Yaskawa INFORM job: SKRZYNIA_5340_90_STOPNI_20BR_OLD.JBI

/JOB
//NAME SKRZYNIA_5340_90_STOPNI_20BR_OLD
///FOLDERNAME 02-SKRZYNIE_JOBS
//POS
///NPOS 552,552,0,39,0,0
///TOOL 0
///POSTYPE PULSE
///PULSE
C00000=0,-52280,40443,0,6876,0
C00001=82314,-24956,17040,59626,-27382,6248
C00002=93910,-8625,17040,59626,-43355,6248
C00003=98846,-1061,-42166,80308,-57081,-16120
C00004=100452,6057,-48127,85711,-56704,-21322
C00005=95573,33077,-33257,84645,-64023,-26851
C00006=94102,33899,-31937,85246,-63371,-26689
C00007=95573,33077,-33257,84645,-64023,-26851
C00008=94862,31071,-36438,85313,-63677,-27192
C00009=95573,33077,-33257,84645,-64023,-26851
C00010=95263,33142,-33256,84677,-63995,-26850
C00011=95263,33142,-33256,84677,-63995,-26850
C00012=94017,33843,-32133,85187,-63445,-26710
C00013=95557,35310,-29762,82906,-65354,-26497
C00014=95275,35582,-29321,82044,-66131,-26480
C00015=95263,33142,-33256,84677,-63995,-26850
C00016=95260,33144,-33256,84678,-63995,-26850
C00017=95260,33144,-33256,84678,-63995,-26850
C00018=94022,33838,-32141,85183,-63448,-26711
C00019=95260,33144,-33256,84678,-63995,-26850
C00020=94618,31343,-36117,85281,-63684,-27157
C00021=95260,33144,-33256,84678,-63995,-26850
C00022=95258,25631,32269,66559,-75499,-2416
C00023=95258,25631,32269,66559,-75499,-2416
C00024=94181,26497,33533,66410,-74896,-2191
C00025=95658,30184,39035,66708,-78559,-2356
C00026=95217,30377,39331,66881,-79841,-2558
C00027=95258,25631,32269,66559,-75499,-2416
C00028=98811,21047,-15512,99242,-81394,-20987
C00029=98811,21047,-15512,99242,-81394,-20987
C00030=97775,21639,-14693,99563,-80753,-20993
C00031=98811,21047,-15512,99242,-81394,-20987
C00032=98206,18840,-18520,99489,-81124,-21211
C00033=98811,21047,-15512,99242,-81394,-20987
C00034=98765,34858,63506,90961,-74847,-417
C00035=98765,34858,63506,90961,-74847,-417
C00036=97741,35895,65220,90657,-74158,-246
C00037=98765,34858,63506,90961,-74847,-417
C00038=98337,32226,59232,91111,-74633,-884
C00039=98765,34858,63506,90961,-74847,-417
C00040=98728,21792,17445,103800,-78809,-12049
C00041=97232,27021,37502,101932,-75086,-7690
C00042=96358,27701,38514,101868,-74464,-7680
C00043=97232,27021,37502,101932,-75086,-7690
C00044=96733,24820,34282,102049,-74905,-7989
C00045=97232,27021,37502,101932,-75086,-7690
C00046=94428,854,16076,89248,-50738,-4740
C00047=88080,-20128,-3199,80943,-31244,-2335
C00048=48287,-44591,-17414,16172,-14532,25809
C00049=48287,-44591,-17414,16172,-14532,25809
C00050=85348,-13130,13838,41209,-47455,8220
C00051=97395,20012,29210,69700,-74457,-9077
C00052=97055,28839,36684,71776,-79389,-10554
C00053=97055,28839,36684,71776,-79389,-10554
C00054=96058,29646,37897,71666,-78799,-10362
C00055=97055,28839,36684,71776,-79389,-10554
C00056=96570,26659,33451,71832,-78911,-10777
C00057=97055,28839,36684,71776,-79389,-10554
C00058=99123,23256,18377,81563,-78104,3156
C00059=99123,23256,18377,81563,-78104,3156
C00060=98123,23909,19300,81582,-77442,3256
C00061=99123,23256,18377,81563,-78104,3156
C00062=98765,21723,16234,81638,-77830,3017
C00063=99123,23256,18377,81563,-78104,3156
C00064=99222,23346,17795,82202,-78388,4176
C00065=99222,23346,17795,82202,-78388,4176
C00066=98149,24045,18779,82229,-77677,4281
C00067=99222,23346,17795,82202,-78388,4176
C00068=98861,21801,15633,82278,-78114,4033
C00069=99222,23346,17795,82202,-78388,4176
C00070=100468,18781,12295,88713,-76630,3899
C00071=100488,13084,3722,91602,-74275,2573
C00072=99329,-2479,-35949,113241,-72472,-2557
C00073=60067,-64368,-72505,144806,-26050,-19168
C00074=60067,-50244,-32501,110603,-14199,-2207
C00075=63330,-26972,24478,18707,-56801,31483
C00076=95462,-32664,-40336,69376,-39980,4046
C00077=97787,-9790,-26685,81509,-54738,-4408
C00078=99864,21793,7359,80466,-76601,-6182
C00079=99862,21793,7358,80466,-76600,-6182
C00080=98290,21024,6297,80683,-75539,-6194
C00081=97471,21541,7008,80756,-75007,-6115
C00082=98290,21024,6297,80683,-75539,-6194
C00083=97834,19245,3873,80814,-75197,-6333
C00084=98290,21024,6297,80683,-75539,-6194
C00085=98946,26804,31705,85784,-78857,-1423
C00086=98946,26804,31705,85784,-78857,-1423
C00087=98292,27270,32391,85749,-78414,-1361
C00088=98946,26804,31705,85784,-78857,-1423
C00089=98631,25349,29587,85839,-78632,-1590
C00090=98946,26804,31705,85784,-78857,-1423
C00091=97031,6331,9149,87487,-63868,-1924
C00092=73503,-30722,-22703,70949,-18863,5788
C00093=42754,-66126,12236,-1301,3231,7194
C00094=0,-52280,40443,0,6876,0
C00095=0,-52280,40443,0,6876,0
C00096=48041,-29633,723,44271,-15597,-57965
C00097=50268,-18118,11295,51661,-15759,-61288
C00098=49280,-17155,12057,50642,-15139,-60911
C00099=50435,-16984,12194,52574,-15707,-61719
C00100=49536,-18455,11034,50297,-15435,-60714
C00101=49756,-19891,11927,46282,-16637,-58724
C00102=49756,-15074,24021,36925,-20097,-54095
C00103=49264,-12389,27117,35970,-20004,-53698
C00104=48191,-11316,28046,34492,-19486,-53134
C00105=50556,-10584,28692,38442,-20269,-54728
C00106=49756,-15074,24021,36925,-20097,-54095
C00107=50509,-14376,22441,40930,-19158,-55976
C00108=50873,-17966,11417,52677,-16048,-61710
C00109=49459,-16590,12517,51258,-15158,-61190
C00110=50592,-16429,12648,53120,-15720,-61960
C00111=50873,-17966,11417,52677,-16048,-61710
C00112=50703,-18403,11066,52155,-16024,-61477
C00113=50703,-18403,11066,52155,-16024,-61477
C00114=49026,-16768,12358,50435,-14971,-60844
C00115=50653,-16371,12680,53228,-15754,-62008
C00116=50703,-18403,11066,52155,-16024,-61477
C00117=50704,-18401,11069,52157,-16021,-61478
C00118=50704,-20525,5414,58956,-14779,-64789
C00119=49025,-18889,6668,57745,-13658,-64384
C00120=50799,-18420,7036,60610,-14610,-65581
C00121=50704,-20525,5414,58956,-14779,-64789
C00122=51005,-17995,11387,52847,-16122,-61778
C00123=51005,-17995,11387,52847,-16122,-61778
C00124=49564,-16598,12501,51417,-15218,-61257
C00125=50954,-16306,12737,53719,-15902,-62212
C00126=51005,-17995,11387,52847,-16122,-61778
C00127=51030,-17981,11395,52891,-16138,-61796
C00128=51030,-17981,11395,52891,-16138,-61796
C00129=49401,-16396,12662,51265,-15114,-61201
C00130=50908,-16047,12947,53789,-15850,-62250
C00131=51030,-17981,11395,52891,-16138,-61796
C00132=50945,-18019,11363,52741,-16103,-61737
C00133=50945,-16980,14081,49884,-16761,-60338
C00134=49117,-15186,15539,47848,-15653,-59576
C00135=50939,-14679,15960,50992,-16487,-60881
C00136=50945,-18019,11363,52741,-16103,-61737
C00137=50945,-18019,11363,52741,-16103,-61737
C00138=50945,-18556,9943,54337,-15776,-62517
C00139=48967,-16606,11493,52445,-14510,-61829
C00140=51083,-15952,12027,56053,-15559,-63336
C00141=50945,-18556,9943,54337,-15776,-62517
C00142=50945,-18019,11363,52741,-16103,-61737
C00143=51350,-15183,18375,46705,-17991,-58719
C00144=49319,-13187,20053,44263,-16830,-57796
C00145=51236,-12618,20544,47529,-17647,-59142
C00146=51350,-15183,18375,46705,-17991,-58719
C00147=50028,-23690,-6096,22921,-31075,-54538
C00148=50670,-23735,-6923,24003,-30760,-55076
C00149=48518,-21492,-5254,21861,-29696,-54082
C00150=50138,-21068,-4928,23831,-30039,-55022
C00151=50670,-23735,-6923,24003,-30760,-55076
C00152=49763,-24225,-29961,22080,-30065,-59113
C00153=49763,-24225,-29961,22080,-30065,-59113
C00154=47727,-21550,-27874,20313,-29013,-58119
C00155=49271,-21042,-27466,22016,-29310,-59069
C00156=49763,-24225,-29961,22080,-30065,-59113
C00157=50713,-12366,-58367,41124,-17813,-74400
C00158=50713,-12366,-58367,41124,-17813,-74400
C00159=48934,-9522,-55687,39981,-16902,-73526
C00160=50242,-8975,-55157,41389,-17374,-74448
C00161=50713,-12366,-58367,41124,-17813,-74400
C00162=49763,-25421,-36239,24565,-26935,-60445
C00163=43547,-31626,-19626,5157,-49140,-52118
C00164=40154,-51179,-915,24203,-8234,-36524
C00165=0,-52280,40443,0,6876,0
C00166=0,-52280,40443,0,6876,0
C00167=2117,-50103,-33543,4117,45077,-85249
C00168=-26439,-48928,-33543,4117,-52362,-85249
C00169=-1453,-29933,-32011,46693,-66666,-90474
C00170=24798,-19255,-10490,69050,-85424,-90395
C00171=18386,-22028,-12683,68302,-81515,-89477
///LIMIT ON
C00172=9843,-31743,-57176,61611,-65235,-99401
C00173=-39603,-23393,-71448,91573,-31907,-107123
C00174=-35705,5077,-63140,100511,-35979,-118164
C00175=-33789,12193,-59259,102607,-37482,-119984
C00176=-34998,13124,-58049,103267,-36945,-119997
C00177=-34401,14597,-56112,102586,-37131,-119778
C00178=-34998,13124,-58049,103267,-36945,-119997
C00179=-36388,13885,-57049,104079,-36338,-120048
C00180=-34998,13124,-58049,103267,-36945,-119997
C00181=-34008,-7969,-75285,118537,-50852,-116988
C00182=-26318,8527,-57077,128458,-81874,-108613
///LIMIT OFF
C00183=-23139,-1795,-12064,73373,-53703,-87448
C00184=-27830,-667,-10848,73187,-50621,-86997
C00185=-27373,916,-9115,73207,-50922,-87041
C00186=-27830,-667,-10848,73187,-50621,-86997
C00187=-28901,-207,-10348,73132,-49918,-86888
C00188=-27830,-667,-10848,73187,-50621,-86997
C00189=-37166,8347,13175,41366,-53536,-76331
C00190=-37403,7707,12401,41298,-53388,-76282
C00191=-36830,9273,14303,41455,-53750,-76396
C00192=-37403,7707,12401,41298,-53388,-76282
C00193=-38235,8246,13056,40951,-53040,-76025
C00194=-37403,7707,12401,41298,-53388,-76282
C00195=-30063,5992,18551,55847,-56234,-77619
C00196=-30754,7414,19761,55747,-55713,-77591
C00197=-30376,8670,21285,55817,-55984,-77619
C00198=-30754,7414,19761,55747,-55713,-77591
C00199=-31265,7672,20073,55566,-55435,-77478
C00200=-30085,6037,18588,55845,-56218,-77619
C00201=-25385,-1715,-9470,94765,-53990,-89712
C00202=-25885,-764,-8323,94779,-53645,-89697
C00203=-25564,418,-7032,94741,-53861,-89683
C00204=-25885,-764,-8323,94779,-53645,-89697
C00205=-26741,-428,-7957,94890,-53068,-89741
C00206=-25421,-1648,-9389,94767,-53966,-89710
C00207=-17789,-39335,-40320,90232,-41783,-86178
C00208=-25885,-761,-8324,94780,-53645,-89696
C00209=-25885,-761,-8324,94780,-53645,-89696
C00210=-25612,239,-7230,94748,-53828,-89684
C00211=-25885,-761,-8324,94780,-53645,-89696
C00212=-26712,-436,-7972,94885,-53087,-89742
C00213=-25885,-761,-8324,94780,-53645,-89696
C00214=-26038,-1317,-8919,94796,-53541,-89701
C00215=-18430,-29121,-33898,93348,-44706,-88207
C00216=-3209,-48313,-44409,84985,-37126,-83197
C00217=-3617,-53456,-46461,81793,-37023,-81323
C00218=-28991,-22310,-29554,94749,-46554,-89251
C00219=-30664,-6343,-14094,96248,-45630,-90223
C00220=-30664,-6343,-14094,96248,-45630,-90223
C00221=-30207,-5031,-12762,96238,-45949,-90236
C00222=-30664,-6343,-14094,96248,-45630,-90223
C00223=-31510,-5971,-13720,96406,-45066,-90297
C00224=-29506,-9179,-17232,96085,-46411,-90159
C00225=-30003,-8487,-16482,96169,-46079,-90194
C00226=-30881,-6301,-14053,96286,-45485,-90239
C00227=-30407,-4956,-12684,96275,-45813,-90252
C00228=-30881,-6301,-14053,96286,-45485,-90239
C00229=-31646,-5963,-13712,96429,-44974,-90305
C00230=-29893,-8752,-16772,96152,-46152,-90188
C00231=-30350,-7636,-15544,96220,-45845,-90215
C00232=-30881,-6301,-14053,96286,-45485,-90239
C00233=-30396,-4924,-12652,96275,-45822,-90251
C00234=-30881,-6301,-14053,96286,-45485,-90239
C00235=-31665,-5954,-13703,96434,-44961,-90308
C00236=-29959,-8593,-16598,96162,-46108,-90192
C00237=-26558,-19284,-27675,95285,-48332,-89713
C00238=-5136,-57382,-50746,80999,-31115,-81799
C00239=-5136,-57382,-50746,80999,-31115,-81799
C00240=-22762,-12288,-20025,94001,-55646,-89200
C00241=-24763,-3131,-11201,94769,-54426,-89746
C00242=-26203,-419,-7954,94818,-53430,-89712
C00243=-25939,548,-6896,94784,-53609,-89698
C00244=-26203,-419,-7954,94818,-53430,-89712
C00245=-26818,-174,-7689,94897,-53016,-89744
C00246=-24998,-2701,-10694,94780,-54264,-89743
C00247=-23275,-722,28392,94611,-50650,-77911
C00248=-21733,-16242,25206,75334,-39210,-63099
C00249=0,-52280,40443,0,6876,0
C00250=0,-52280,40443,0,6876,0
C00251=82314,-24956,17040,59626,-27382,6248
C00252=93910,-8625,17040,59626,-43355,6248
C00253=98846,-1061,-42166,80308,-57081,-16120
C00254=100452,6057,-48127,85711,-56704,-21322
C00255=95564,34698,-34234,85516,-63941,-27819
C00256=93687,36612,-31081,84292,-64733,-27467
C00257=93711,36598,-31105,84282,-64744,-27471
C00258=95564,34698,-34234,85516,-63941,-27819
C00259=96930,32282,-32252,82595,-65816,-26305
C00260=93663,32611,-31732,84127,-64318,-26195
C00261=93663,32611,-31732,84127,-64318,-26195
C00262=96930,32282,-32252,82595,-65816,-26305
C00263=96528,-7533,-34932,76119,-53878,-10439
C00264=88377,-34186,-45291,67238,-52212,-2442
C00265=73560,-62084,7826,28695,-34737,3666
C00266=0,-52280,40443,0,6876,0
C00267=0,-52280,40443,0,6876,0
C00268=2117,-50103,-33543,4117,45077,-85249
C00269=-26439,-48928,-33543,4117,-52362,-85249
C00270=-26439,-27355,-33543,41485,-52362,-85249
C00271=-39218,-24492,-41653,51934,-39374,-86964
C00272=-37997,-10433,-19136,70610,-34172,-88069
C00273=-38397,-8978,-17736,70703,-33874,-88109
C00274=-39218,-24492,-41653,51934,-39374,-86964
C00275=-26439,-27355,-33543,41485,-52362,-85249
C00276=1598,-24403,-16502,45671,-72599,-88798
C00277=-11365,-15171,10010,30164,-77975,-82960
C00278=-38112,4197,-14374,43778,-42973,-90436
C00279=-39116,7904,-10019,43942,-43580,-90646
C00280=-38495,8531,-9262,44482,-44499,-91194
C00281=-38112,4197,-14374,43778,-42973,-90436
C00282=-53220,-12364,-8957,19277,-47766,-73858
C00283=-11365,-15171,10010,30164,-77975,-82960
C00284=-16156,-38280,11293,23671,-42998,-42040
C00285=-11365,-47379,10010,30164,3063,-681
C00286=0,-52280,40443,0,6876,0
C00287=0,-36700,24612,-42871,-31823,-33862
C00288=44403,-30110,7154,24155,-23805,-45557
C00289=51347,-17798,16373,37641,-23556,-51399
C00290=51570,-17239,16856,38066,-23574,-51584
C00291=66077,-16287,3920,86568,-32028,-80947
C00292=60657,-14974,12588,70166,-26612,-71053
C00293=40431,-28773,9158,17648,-23273,-42875
C00294=0,-36700,24612,-42871,-31823,-33862
C00295=0,-52280,40443,0,6876,0
C00296=0,-52280,40443,0,6876,0
C00297=73560,-62084,7826,28695,-34737,3666
C00298=88377,-34186,-45291,67238,-52212,-2442
C00299=96528,-7533,-34932,76119,-53878,-10439
C00300=100432,21324,12575,83706,-77956,-7498
C00301=100432,21324,12575,83706,-77956,-7498
C00302=97224,21170,12361,83970,-75786,-7447
C00303=97224,21170,12361,83970,-75786,-7447
C00304=100432,21324,12575,83706,-77956,-7498
C00305=100432,21324,12575,83706,-77956,-7498
C00306=97481,25108,17890,83512,-78432,-7131
C00307=97624,25049,17805,83504,-78528,-7141
C00308=100432,21324,12575,83706,-77956,-7498
C00309=97137,1790,-11103,86179,-63102,-7963
C00310=99183,2264,5333,86781,-62651,-3264
C00311=99868,-33,22146,72719,-59601,5126
C00312=99028,-10516,17309,71061,-60695,4227
C00313=58820,-39124,10926,53325,-41870,3759
C00314=0,-52280,40443,0,6876,0
C00315=37281,-50778,-9546,79570,-75313,-71156
C00316=21038,-23698,-30323,82948,-81132,-85647
C00317=-27256,-5882,-14331,85818,-48304,-85968
C00318=-24751,2890,-4920,85349,-55822,-86178
C00319=-24793,2953,-4845,85351,-55796,-86173
C00320=-27256,-5882,-14331,85818,-48304,-85968
C00321=-21143,-15675,-23596,84785,-52496,-85466
C00322=35274,-15248,-23220,82440,-90817,-86704
C00323=35274,-15248,-23220,82440,-90817,-86704
C00324=-45551,161,-18089,35087,-36064,-73293
C00325=-42435,6767,-10562,40540,-41185,-77662
C00326=-42821,6494,-10882,40094,-40673,-77276
C00327=-45551,161,-18089,35087,-36064,-73293
C00328=-32891,-7184,-22739,69075,-41395,-83248
C00329=-29265,-39765,-39402,58096,-43152,-73226
C00330=-37287,-55159,35520,2191,5667,-2084
C00331=0,-52280,40443,0,6876,0
C00332=0,-36700,24612,-42871,-31823,-33862
C00333=44403,-30110,7154,24155,-23805,-45557
C00334=44403,-30110,7154,24155,-23805,-45557
C00335=42101,-12213,25656,103795,-5192,-78630
C00336=46259,-8171,27719,110365,-8144,-81138
C00337=52601,-3768,32601,101908,-15442,-75329
C00338=55043,-3560,27637,120535,-21833,-87376
C00339=55127,-3656,27536,120476,-21875,-87335
C00340=50677,-23266,8367,38735,-22212,-52049
C00341=47073,-34549,9488,27883,-30316,-51458
C00342=0,-52280,40443,0,6876,0
C00343=0,-52280,40443,0,6876,0
C00344=73560,-62084,7826,28695,-34737,3666
C00345=96983,-27116,-23481,78724,-62297,-1998
C00346=100467,-7393,-15195,81625,-60158,-6002
C00347=99336,18440,8642,84276,-74234,-7647
C00348=99336,18440,8642,84276,-74234,-7647
C00349=97735,24994,14595,85350,-78994,-5109
C00350=97744,25074,13580,86004,-79195,-4385
C00351=99336,18440,8642,84276,-74234,-7647
C00352=99336,18440,8642,84276,-74234,-7647
C00353=97891,23737,8261,88167,-79183,-2386
C00354=97851,23541,8142,88101,-79081,-2507
C00355=99336,18440,8642,84276,-74234,-7647
C00356=89817,-17341,-38408,97132,-45323,-12250
C00357=100347,-21961,-42251,93939,-52125,-11121
C00358=60204,-59872,-73451,117647,-17639,-18840
C00359=37721,-67612,11381,1325,-438,7850
C00360=-37287,-55159,35520,2191,5667,-2084
C00361=-40042,-68802,-18337,47708,-19461,-45384
C00362=-28646,-23138,-32952,89786,-42552,-85395
C00363=-38882,-16596,-17625,44304,-41043,-72768
C00364=-42680,-6319,-12818,46127,-36112,-73823
C00365=-37459,704,-5408,52536,-43357,-78192
C00366=-32778,4349,-7465,59128,-48375,-83352
C00367=-42680,-6319,-12818,46127,-36112,-73823
C00368=-38882,-16596,-17625,44304,-41043,-72768
C00369=-28646,-23138,-32952,89786,-42552,-85395
C00370=-29905,-15291,-26411,91102,-43435,-86304
C00371=-25469,1350,-9790,89991,-54827,-86555
C00372=-24242,3379,-7505,89554,-57286,-86471
C00373=-29905,-15291,-26411,91102,-43435,-86304
C00374=-40042,-68802,-18337,47708,-19461,-45384
C00375=-37287,-55159,35520,2191,5667,-2084
C00376=0,-52280,40443,0,6876,0
C00377=37164,-60659,6466,13301,-5027,-19773
C00378=45362,-39990,2831,27538,-17767,-40935
C00379=57189,-26834,-7130,38780,-31731,-51561
C00380=63456,-14144,8594,45591,-40850,-50620
C00381=63298,-23815,-40708,66066,-30898,-63274
C00382=57189,-26834,-7130,38780,-31731,-51561
C00383=41180,-61187,4729,17280,-8498,-23442
C00384=0,-52280,40443,0,6876,0
C00385=0,-52280,40443,0,6876,0
C00386=37721,-67612,11381,1325,-438,7850
C00387=43180,-50572,-20637,6552,-29302,38834
C00388=95618,-29588,-12765,65168,-50072,21743
C00389=-36913,-32963,-979,75363,-26772,-58744
C00390=-42264,1508,8544,35869,-47237,-69477
C00391=-43183,4597,12058,35318,-46938,-69128
C00392=-43183,5775,16318,34276,-48598,-68388
C00393=-42264,1508,8544,35869,-47237,-69477
C00394=56258,-38103,3288,28818,-33580,-23051
C00395=41438,-37635,17580,13151,-29920,-38779
C00396=54964,-26842,8528,44141,-23181,-52038
C00397=50761,-21373,7883,46957,-18149,-54038
C00398=65037,-17203,-4749,103175,-32218,-89355
C00399=65312,-6152,27526,81270,-31139,-77237
C00400=56762,-20631,11812,69834,-24329,-69917
C00401=46096,-45842,-2681,20981,-19497,-36310
C00402=41180,-61187,4729,17280,-8498,-23442
C00403=0,-52280,40443,0,6876,0
C00404=0,-52280,40443,0,6876,0
C00405=37721,-67612,11381,1325,-438,7850
C00406=43180,-50572,-20637,6552,-29302,38834
C00407=79425,-37128,-15462,51820,-35721,18807
C00408=92377,-29666,-26166,73570,-38078,7008
C00409=97441,-6012,-18634,86114,-58345,-2339
C00410=98864,-2001,-14672,90389,-62789,-3799
C00411=98767,21176,13691,87588,-77304,-2577
C00412=98123,23617,17097,87345,-78645,-2335
C00413=97979,23711,17231,87352,-78549,-2326
C00414=98995,11633,1143,88650,-71928,-3309
C00415=98055,11605,-2710,80204,-69934,-2921
C00416=97049,22713,12201,78728,-76277,-2408
C00417=97049,22025,5529,79613,-75682,-4326
C00418=98864,-2001,-14672,90389,-62789,-3799
C00419=100472,-329,-13432,98539,-67097,-6304
C00420=92822,-26306,-37175,103295,-43881,-7703
C00421=68601,-52593,-52127,95725,-25602,-3235
C00422=80632,-38079,-20908,64053,-45216,12949
C00423=43180,-50572,-20637,6552,-29302,38834
C00424=37721,-67612,11381,1325,-438,7850
C00425=0,-52280,40443,0,6876,0
C00426=0,-52280,40443,0,6876,0
C00427=0,-52280,40443,0,-39412,36675
C00428=-54026,-30203,28811,-7745,-28969,-5087
C00429=-30389,-9386,-5824,79667,-43789,-73484
C00430=-32979,-3325,255,79720,-41988,-73575
C00431=-25304,6223,10893,81656,-55729,-74481
C00432=-23842,8927,14147,81883,-58875,-74544
C00433=-30389,-9386,-5824,79667,-43789,-73484
C00434=-32145,-6440,-2937,79673,-42575,-73527
C00435=-25014,6414,11121,81706,-56254,-74506
C00436=-23603,11547,23533,79434,-59735,-72187
C00437=-32145,-5050,2357,77009,-42992,-71800
C00438=-35251,-18143,20376,53513,-41117,-59413
C00439=-9534,-43450,13514,26959,-29486,-38723
C00440=-22834,-59963,22946,6692,-2150,-9612
C00441=0,-52280,40443,0,6876,0
C00442=23708,-46776,23536,16027,-4787,-19738
C00443=50917,-40459,4132,34421,-18173,-42391
C00444=51059,-36587,4608,36647,-19418,-45358
C00445=50113,-22729,10834,36393,-23396,-50963
C00446=61700,-17481,4291,79414,-27019,-76651
C00447=63551,-15463,7666,79999,-29336,-77075
C00448=50113,-22729,10834,36393,-23396,-50963
C00449=31287,-69981,-10850,7253,-6843,-20996
C00450=19644,-57271,30737,863,5243,-2499
C00451=0,-52280,40443,0,6876,0
C00452=0,-52280,40443,0,6876,0
C00453=37721,-67612,11381,1325,-438,7850
C00454=43180,-50572,-20637,6552,-29302,38834
C00455=79425,-37128,-15462,51820,-35721,18807
C00456=92377,-33385,-41303,83059,-36844,1354
C00457=97439,-6020,-18641,86113,-58338,-2338
C00458=98442,-3149,-15680,86092,-59018,-2413
C00459=96855,-5742,-18360,86176,-57949,-2343
C00460=99185,22470,15697,83135,-77937,-1734
C00461=97717,21807,14770,83256,-76932,-1762
C00462=97717,21807,14770,83256,-76932,-1762
C00463=99185,24652,26607,82087,-78431,1026
C00464=99185,22470,15697,83135,-77937,-1734
C00465=97852,24994,19264,82957,-78889,-1504
C00466=97683,25109,19429,82963,-78778,-1488
C00467=99870,24121,23963,82328,-78767,341
C00468=100471,12680,2182,89317,-73847,-3746
C00469=93923,-8883,-21959,92925,-54783,-4609
C00470=92822,-26306,-37175,103295,-43881,-7703
C00471=68601,-52593,-52127,95725,-25602,-3235
C00472=80632,-38079,-20908,64053,-45216,12949
C00473=43180,-50572,-20637,6552,-29302,38834
C00474=37721,-67612,11381,1325,-438,7850
C00475=0,-52280,40443,0,6876,0
C00476=0,-52280,40443,0,6876,0
C00477=0,-52280,40443,0,-39412,36675
C00478=-54026,-30203,28811,-7745,-28969,-5087
C00479=-81492,-18979,22896,-11682,-23662,-26316
C00480=-32145,-2720,10458,73217,-43826,-69319
C00481=-32145,-2720,10458,73217,-43826,-69319
C00482=-25800,12961,35355,74076,-56913,-68018
C00483=-23961,12723,28512,77913,-59573,-70804
C00484=-32145,-2720,10458,73217,-43826,-69319
C00485=-34274,-9754,-24316,117159,-46217,-86271
C00486=-34274,-9754,-24316,117159,-46217,-86271
C00487=-29822,-1437,-15851,112752,-53901,-84078
C00488=-28945,-336,-14662,112011,-55335,-83695
C00489=-34274,-9754,-24316,117159,-46217,-86271
C00490=-34422,-9999,20796,72411,-42519,-66994
C00491=-35251,-18143,20376,53513,-41117,-59413
C00492=-9534,-43450,13514,26959,-29486,-38723
C00493=-22834,-59963,22946,6692,-2150,-9612
C00494=0,-52280,40443,0,6876,0
C00495=44101,-76445,-48847,15697,-17168,-40457
C00496=49121,-28282,-35458,21895,-29219,-59001
C00497=50484,-13386,-55713,36158,-19724,-71897
C00498=55938,-10187,-55661,55618,-22248,-82832
C00499=57471,15289,-57256,78033,-21049,-89958
C00500=50484,-13386,-55713,36158,-19724,-71897
C00501=49763,-25421,-36239,24565,-26935,-60445
C00502=50529,-22709,-3778,22940,-31995,-54502
C00503=45389,-28224,4312,35967,-15579,-54278
C00504=40154,-51179,-915,24203,-8234,-36524
C00505=0,-52280,40443,0,6876,0
C00506=0,-52280,40443,0,6876,0
C00507=37721,-67612,11381,1325,-438,7850
C00508=43181,-50571,-20637,6551,-29300,38834
C00509=92325,-23846,-7228,63960,-40898,12897
C00510=85237,-2771,25348,50990,-49534,17622
C00511=95240,9110,29862,65614,-64506,10679
C00512=98093,21269,34291,73470,-75068,6437
C00513=97988,24882,21615,85608,-78767,-653
C00514=97988,24882,21615,85608,-78767,-653
C00515=97983,26659,41434,72953,-78426,6910
C00516=99525,21729,17159,85870,-76787,-954
C00517=97991,25479,22462,85564,-79108,-597
C00518=97991,25479,22462,85564,-79108,-597
C00519=99525,21729,17159,85870,-76787,-954
C00520=99266,24955,27205,94359,-77696,-2486
C00521=97188,23163,26035,94281,-76219,-2314
C00522=96376,23467,25710,100017,-76114,-3586
C00523=96491,23385,25594,100018,-76194,-3586
C00524=96491,25838,35147,98979,-75163,-1386
C00525=98212,22329,20183,100499,-78017,-4807
C00526=97122,-3279,-3245,90778,-58787,-678
C00527=97513,-10257,11960,71433,-51152,11355
C00528=72477,-33752,-3372,52810,-39669,19964
C00529=0,-52278,40443,0,6872,5
C00530=0,-52278,40443,31822,-65283,-46097
C00531=-7820,3000,44222,77356,-66876,-70486
C00532=-24244,23423,72059,64993,-61079,-67138
C00533=-27261,30732,84230,62108,-60720,-65392
C00534=-22394,37028,87531,68934,-68535,-64461
C00535=-24244,23423,72059,64993,-61079,-67138
C00536=3014,-20441,-7349,104591,-68614,-79454
C00537=6322,-14118,13197,96169,-69167,-72790
C00538=14133,-16757,18528,88010,-59455,-67296
C00539=-10261,-46634,14475,36899,-22136,-31570
C00540=-22834,-59963,22946,6692,-2150,-9612
C00541=0,-52280,40443,0,6876,0
C00542=23708,-46776,23536,16027,-4787,-19738
C00543=50917,-40459,4132,34421,-18173,-42391
C00544=49876,-21948,7530,68838,-10324,-59148
C00545=46721,-18942,9765,68167,-8197,-59205
C00546=59102,-15651,-1637,118714,-27356,-88041
C00547=59185,-13834,7185,105143,-23914,-78054
C00548=45927,-22803,4403,78462,-8511,-64553
C00549=62498,-35400,-2607,72048,-19281,-59202
C00550=31287,-69981,-10850,7253,-6843,-20996
C00551=0,-52280,40443,0,6876,0
BC00000=487510
BC00001=445130
BC00002=445130
BC00003=445130
BC00004=445130
BC00005=468227
BC00006=468227
BC00007=468227
BC00008=468227
BC00009=468227
BC00010=514421
BC00011=514421
BC00012=514421
BC00013=514421
BC00014=514421
BC00015=514421
BC00016=560588
BC00017=560588
BC00018=560588
BC00019=560588
BC00020=560588
BC00021=560588
BC00022=536404
BC00023=536404
BC00024=536404
BC00025=536404
BC00026=536404
BC00027=536404
BC00028=582458
BC00029=582458
BC00030=582458
BC00031=582458
BC00032=582458
BC00033=582458
BC00034=581206
BC00035=581206
BC00036=581206
BC00037=581206
BC00038=581206
BC00039=581206
BC00040=626960
BC00041=626960
BC00042=626960
BC00043=626960
BC00044=626960
BC00045=626960
BC00046=604255
BC00047=604255
BC00048=604255
BC00049=699121
BC00050=714117
BC00051=772491
BC00052=770398
BC00053=770398
BC00054=770398
BC00055=770398
BC00056=770398
BC00057=770398
BC00058=820815
BC00059=820815
BC00060=820815
BC00061=820815
BC00062=820815
BC00063=820815
BC00064=866263
BC00065=866263
BC00066=866260
BC00067=866263
BC00068=866263
BC00069=866263
BC00070=868226
BC00071=868803
BC00072=869038
BC00073=872244
BC00074=872244
BC00075=929479
BC00076=991951
BC00077=992064
BC00078=992095
BC00079=979853
BC00080=976781
BC00081=976781
BC00082=976781
BC00083=976781
BC00084=976781
BC00085=963886
BC00086=963886
BC00087=963886
BC00088=963886
BC00089=963886
BC00090=963886
BC00091=965124
BC00092=964905
BC00093=857759
BC00094=811793
BC00095=811793
BC00096=953382
BC00097=953382
BC00098=953382
BC00099=953382
BC00100=953382
BC00101=953382
BC00102=983298
BC00103=983298
BC00104=983298
BC00105=983298
BC00106=983298
BC00107=865016
BC00108=888056
BC00109=888056
BC00110=888056
BC00111=888056
BC00112=830714
BC00113=830714
BC00114=830714
BC00115=830714
BC00116=830714
BC00117=764829
BC00118=764829
BC00119=764829
BC00120=764829
BC00121=764829
BC00122=707174
BC00123=707174
BC00124=707174
BC00125=707174
BC00126=707174
BC00127=642071
BC00128=642071
BC00129=642071
BC00130=642071
BC00131=642071
BC00132=584746
BC00133=584746
BC00134=584746
BC00135=584746
BC00136=584746
BC00137=519232
BC00138=519232
BC00139=519232
BC00140=519232
BC00141=519232
BC00142=461813
BC00143=461813
BC00144=461813
BC00145=461813
BC00146=461813
BC00147=459544
BC00148=459544
BC00149=459544
BC00150=459544
BC00151=459544
BC00152=459544
BC00153=459544
BC00154=459544
BC00155=459544
BC00156=459544
BC00157=459544
BC00158=459544
BC00159=459544
BC00160=459544
BC00161=459544
BC00162=459544
BC00163=462325
BC00164=533216
BC00165=533216
BC00166=492150
BC00167=423885
BC00168=423885
BC00169=519103
BC00170=542802
BC00171=634915
BC00172=493160
BC00173=493160
BC00174=517936
BC00175=517447
BC00176=516208
BC00177=516208
BC00178=516208
BC00179=516208
BC00180=516208
BC00181=525487
BC00182=485388
BC00183=500803
BC00184=500803
BC00185=500803
BC00186=500803
BC00187=500803
BC00188=500803
BC00189=585253
BC00190=585253
BC00191=585253
BC00192=585253
BC00193=585253
BC00194=585253
BC00195=600589
BC00196=600589
BC00197=600589
BC00198=600589
BC00199=600589
BC00200=600589
BC00201=646713
BC00202=646713
BC00203=646713
BC00204=646713
BC00205=646713
BC00206=646713
BC00207=659006
BC00208=692822
BC00209=692822
BC00210=692822
BC00211=692822
BC00212=692822
BC00213=692822
BC00214=669701
BC00215=669701
BC00216=669701
BC00217=791136
BC00218=762000
BC00219=762000
BC00220=762000
BC00221=762000
BC00222=762000
BC00223=762000
BC00224=762000
BC00225=831025
BC00226=831025
BC00227=831025
BC00228=831025
BC00229=831025
BC00230=831025
BC00231=877128
BC00232=877128
BC00233=877128
BC00234=877128
BC00235=877128
BC00236=877128
BC00237=854090
BC00238=854090
BC00239=990684
BC00240=992363
BC00241=992364
BC00242=992364
BC00243=992364
BC00244=992364
BC00245=992364
BC00246=992364
BC00247=941750
BC00248=932032
BC00249=771415
BC00250=445130
BC00251=445130
BC00252=445130
BC00253=445130
BC00254=445130
BC00255=475938
BC00256=475938
BC00257=468314
BC00258=475938
BC00259=515329
BC00260=515329
BC00261=507641
BC00262=515329
BC00263=542207
BC00264=542207
BC00265=542207
BC00266=542207
BC00267=492150
BC00268=423885
BC00269=423885
BC00270=423885
BC00271=423885
BC00272=406365
BC00273=406365
BC00274=423885
BC00275=423885
BC00276=423885
BC00277=423885
BC00278=507950
BC00279=507950
BC00280=500226
BC00281=507950
BC00282=493160
BC00283=493160
BC00284=493160
BC00285=493160
BC00286=493160
BC00287=582810
BC00288=655182
BC00289=712102
BC00290=712780
BC00291=712780
BC00292=769565
BC00293=773753
BC00294=582810
BC00295=493160
BC00296=542207
BC00297=542207
BC00298=542207
BC00299=590944
BC00300=543764
BC00301=459277
BC00302=459277
BC00303=451665
BC00304=459277
BC00305=520748
BC00306=520748
BC00307=528468
BC00308=520748
BC00309=524597
BC00310=604006
BC00311=584417
BC00312=584417
BC00313=584417
BC00314=584417
BC00315=542360
BC00316=521200
BC00317=474976
BC00318=474976
BC00319=482600
BC00320=474976
BC00321=474976
BC00322=474976
BC00323=630364
BC00324=628593
BC00325=624867
BC00326=617183
BC00327=631527
BC00328=617183
BC00329=617427
BC00330=620193
BC00331=620193
BC00332=812803
BC00333=887783
BC00334=927066
BC00335=893694
BC00336=914884
BC00337=914884
BC00338=958625
BC00339=987905
BC00340=962387
BC00341=853059
BC00342=542207
BC00343=542207
BC00344=542207
BC00345=541760
BC00346=590944
BC00347=571989
BC00348=566860
BC00349=566868
BC00350=574636
BC00351=566860
BC00352=635958
BC00353=635958
BC00354=643642
BC00355=635958
BC00356=635118
BC00357=635118
BC00358=656468
BC00359=665809
BC00360=620193
BC00361=620193
BC00362=635598
BC00363=635598
BC00364=635598
BC00365=635598
BC00366=635598
BC00367=635598
BC00368=635598
BC00369=635598
BC00370=658627
BC00371=658627
BC00372=666320
BC00373=658627
BC00374=620193
BC00375=620193
BC00376=620193
BC00377=561542
BC00378=498768
BC00379=452071
BC00380=452071
BC00381=452075
BC00382=452071
BC00383=524165
BC00384=524165
BC00385=733103
BC00386=733103
BC00387=733103
BC00388=615413
BC00389=696009
BC00390=735643
BC00391=735643
BC00392=739967
BC00393=735643
BC00394=617218
BC00395=582869
BC00396=580754
BC00397=589556
BC00398=589556
BC00399=626883
BC00400=634257
BC00401=536572
BC00402=561088
BC00403=547800
BC00404=733103
BC00405=733103
BC00406=733103
BC00407=733103
BC00408=733103
BC00409=750523
BC00410=740531
BC00411=740531
BC00412=740531
BC00413=748211
BC00414=744786
BC00415=744786
BC00416=744786
BC00417=744786
BC00418=740531
BC00419=750469
BC00420=750469
BC00421=750469
BC00422=783373
BC00423=795297
BC00424=733103
BC00425=733103
BC00426=672709
BC00427=672709
BC00428=762701
BC00429=743900
BC00430=736524
BC00431=736351
BC00432=743900
BC00433=743900
BC00434=759331
BC00435=759331
BC00436=759331
BC00437=759331
BC00438=750104
BC00439=672725
BC00440=672725
BC00441=672725
BC00442=766882
BC00443=791101
BC00444=802867
BC00445=836517
BC00446=836517
BC00447=894876
BC00448=836517
BC00449=618402
BC00450=618402
BC00451=618402
BC00452=733103
BC00453=733103
BC00454=837215
BC00455=821905
BC00456=831485
BC00457=838453
BC00458=815683
BC00459=817504
BC00460=817504
BC00461=817504
BC00462=825298
BC00463=817504
BC00464=863642
BC00465=863642
BC00466=871437
BC00467=863642
BC00468=817424
BC00469=817332
BC00470=750469
BC00471=750469
BC00472=783373
BC00473=795297
BC00474=733103
BC00475=733103
BC00476=672709
BC00477=672709
BC00478=762701
BC00479=791880
BC00480=819491
BC00481=819491
BC00482=817331
BC00483=817331
BC00484=817326
BC00485=863478
BC00486=863478
BC00487=863478
BC00488=871062
BC00489=863478
BC00490=774095
BC00491=750104
BC00492=672725
BC00493=672725
BC00494=672725
BC00495=528256
BC00496=459544
BC00497=459544
BC00498=459544
BC00499=459547
BC00500=459544
BC00501=459544
BC00502=459544
BC00503=459540
BC00504=533216
BC00505=533216
BC00506=733103
BC00507=733103
BC00508=958571
BC00509=956295
BC00510=943703
BC00511=958036
BC00512=967318
BC00513=947035
BC00514=954731
BC00515=973151
BC00516=970062
BC00517=970062
BC00518=977728
BC00519=978768
BC00520=1019602
BC00521=1018002
BC00522=1016590
BC00523=1035130
BC00524=1035130
BC00525=1019602
BC00526=991903
BC00527=955597
BC00528=952322
BC00529=852584
BC00530=921533
BC00531=958534
BC00532=946591
BC00533=946591
BC00534=946592
BC00535=954904
BC00536=963295
BC00537=934184
BC00538=908449
BC00539=754884
BC00540=672725
BC00541=672725
BC00542=562340
BC00543=452362
BC00544=452362
BC00545=452362
BC00546=452362
BC00547=513216
BC00548=512110
BC00549=512008
BC00550=742282
BC00551=742282
///POSTYPE BASE
///RECTAN
///RCONF 0,0,0,0,0,0,0,0,0,0,0,0,0,0,0,0,0,0,0,0,0,0,0,0
P00006=-2.449,0.031,8.825,0.0000,0.0000,0.0000
P00058=0.000,0.000,3.000,0.0000,0.0000,0.0000
///RCONF 1,0,0,0,0,0,0,0,0,0,0,0,0,0,0,0,0,0,0,0,0,0,0,0
P00300=-0.036,-1.505,2.318,0.0000,0.0000,0.0000
///RCONF 0,0,0,0,0,0,0,0,0,0,0,0,0,0,0,0,0,0,0,0,0,0,0,0
P00301=0.005,-4.708,-4.628,0.0000,0.0000,0.0000
P00302=0.052,-2.937,-4.426,0.0000,0.0000,0.0000
P00303=-0.004,-1.437,-4.584,0.0000,0.0000,0.0000
P00304=0.028,-1.666,-4.234,0.0000,0.0000,0.0000
P00305=-0.003,-1.920,-3.501,0.0000,0.0000,0.0000
P00306=0.015,-2.252,-3.054,0.0000,0.0000,0.0000
P00307=0.019,-2.151,-5.077,0.0000,0.0000,0.0000
P00308=-0.003,-2.092,-4.888,0.0000,0.0000,0.0000
P00309=-0.040,-2.205,-4.992,0.0000,0.0000,0.0000
P00310=-0.006,-2.490,-5.925,0.0000,0.0000,0.0000
P00311=-0.007,-2.079,-5.307,0.0000,0.0000,0.0000
///RCONF 1,0,0,0,0,0,0,0,0,0,0,0,0,0,0,0,0,0,0,0,0,0,0,0
P00349=0.060,0.167,-1.133,0.0000,0.0000,0.0000
///RCONF 0,0,0,0,0,0,0,0,0,0,0,0,0,0,0,0,0,0,0,0,0,0,0,0
P00350=11.519,-0.008,1.149,0.0000,0.0000,0.0000
P00351=13.563,-0.027,-0.653,0.0000,0.0000,0.0000
P00352=13.252,-0.027,-0.827,0.0000,0.0000,0.0000
P00353=10.971,-0.082,0.776,0.0000,0.0000,0.0000
P00354=-0.024,2.508,-1.824,0.0000,0.0000,0.0000
P00355=-0.001,2.528,-1.131,0.0000,0.0000,0.0000
P00356=-0.034,2.921,-0.262,0.0000,0.0000,0.0000
P00357=0.003,3.386,-0.091,0.0000,0.0000,0.0000
P00358=0.014,3.037,-0.020,0.0000,0.0000,0.0000
P00359=-0.005,2.731,0.912,0.0000,0.0000,0.0000
P00360=-0.011,3.412,0.438,0.0000,0.0000,0.0000
P00361=0.018,3.050,1.253,0.0000,0.0000,0.0000
P00400=5.920,-3.503,-0.024,0.0000,0.0000,0.0000
P00401=3.430,-0.021,1.131,0.0000,0.0000,0.0000
P00402=-0.253,1.107,3.062,0.0000,0.0000,0.0000
P00403=-3.666,-0.015,5.328,0.0000,0.0000,0.0000
///RCONF 1,0,0,0,0,0,0,0,0,0,0,0,0,0,0,0,0,0,0,0,0,0,0,0
P00404=0.029,4.189,-1.030,0.0000,0.0000,0.0000
///RCONF 0,0,0,0,0,0,0,0,0,0,0,0,0,0,0,0,0,0,0,0,0,0,0,0
P00405=2.420,0.007,1.427,0.0000,0.0000,0.0000
P00406=3.513,-0.022,0.429,0.0000,0.0000,0.0000
///RCONF 1,0,0,0,1,0,0,0,0,0,0,0,0,0,0,0,0,0,0,0,0,0,0,0
P00407=-0.029,2.348,-1.469,0.0000,0.0000,0.0000
P00408=0.010,1.346,-1.479,0.0000,0.0000,0.0000
///RCONF 1,0,0,0,0,0,0,0,0,0,0,0,0,0,0,0,0,0,0,0,0,0,0,0
P00409=-0.026,2.090,-1.483,0.0000,0.0000,0.0000
P00410=0.001,4.491,-0.583,0.0000,0.0000,0.0000
///RCONF 1,0,0,0,1,0,0,0,0,0,0,0,0,0,0,0,0,0,0,0,0,0,0,0
P00411=-0.015,3.627,0.872,0.0000,0.0000,0.0000
//INST
///DATE 2024/12/20 08:55
///ATTR SC,RW
///GROUP1 RB1,BS1
NOP
CALL JOB:MOVE_INTO_TUNNEL
MOVJ C00000 BC00000 VJ=10.00
MOVJ C00001 BC00001 VJ=30.00
MOVJ C00002 BC00002 VJ=30.00
MOVL C00003 BC00003 V=500.0
MOVJ C00004 BC00004 VJ=30.00
'------------------------
'W65.3
'------------------------
MOVL C00005 BC00005 V=333.3 PL=0
REFP 3 C00006 BC00006
CALL JOB:SEARCH-R1
SET P0300 P0006
SFTON P0300
MOVL C00007 BC00007 V=333.3 PL=0
REFP 3 C00008 BC00008
CALL JOB:SEARCH-R1
SET P0300 P0006
SFTON P0300
MOVL C00009 BC00009 V=333.3 PL=0
SFTOF
'------------------------
'W65.5
'------------------------
MOVL C00010 BC00010 V=500.0
MOVL C00011 BC00011 V=333.3 PL=0
REFP 3 C00012 BC00012
CALL JOB:SEARCH-R1
SET P0301 P0006
SFTON P0301
MOVL C00013 BC00013 V=333.3 PL=0
REFP 3 C00014 BC00014
CALL JOB:SEARCH-R1
SET P0301 P0006
SFTON P0301
MOVL C00015 BC00015 V=333.3 PL=0
SFTOF
'------------------------
'W65.7
'------------------------
MOVL C00016 BC00016 V=500.0
MOVL C00017 BC00017 V=333.3 PL=0
REFP 3 C00018 BC00018
CALL JOB:SEARCH-R1
SET P0302 P0006
SFTON P0302
MOVL C00019 BC00019 V=333.3 PL=0
REFP 3 C00020 BC00020
CALL JOB:SEARCH-R1
SET P0302 P0006
SFTON P0302
MOVL C00021 BC00021 V=500.0 PL=0
SFTOF
'------------------------
'W65.10
'------------------------
MOVL C00022 BC00022 V=500.0
MOVL C00023 BC00023 V=333.3 PL=0
REFP 3 C00024 BC00024
CALL JOB:SEARCH-R1
SET P0303 P0006
SFTON P0303
MOVL C00025 BC00025 V=333.3 PL=0
REFP 3 C00026 BC00026
CALL JOB:SEARCH-R1
SET P0303 P0006
SFTON P0303
MOVL C00027 BC00027 V=333.3 PL=0
SFTOF
'------------------------
'W65.12
'------------------------
MOVL C00028 BC00028 V=500.0
MOVL C00029 BC00029 V=333.3 PL=0
REFP 3 C00030 BC00030
CALL JOB:SEARCH-R1
SET P0304 P0006
SFTON P0304
MOVL C00031 BC00031 V=333.3 PL=0
REFP 3 C00032 BC00032
CALL JOB:SEARCH-R1
SET P0304 P0006
SFTON P0304
MOVL C00033 BC00033 V=333.3 PL=0
SFTOF
'------------------------
'W65.15
'------------------------
MOVL C00034 BC00034 V=500.0
MOVL C00035 BC00035 V=333.3 PL=0
REFP 3 C00036 BC00036
CALL JOB:SEARCH-R1
SET P0305 P0006
SFTON P0305
MOVL C00037 BC00037 V=333.3 PL=0
REFP 3 C00038 BC00038
CALL JOB:SEARCH-R1
SET P0305 P0006
SFTON P0305
MOVL C00039 BC00039 V=333.3 PL=0
SFTOF
'------------------------
'W65.17
'------------------------
MOVL C00040 BC00040 V=500.0
MOVL C00041 BC00041 V=166.7 PL=0
REFP 3 C00042 BC00042
CALL JOB:SEARCH-R1
SET P0306 P0006
SFTON P0306
MOVL C00043 BC00043 V=333.3 PL=0
REFP 3 C00044 BC00044
CALL JOB:SEARCH-R1
SET P0306 P0006
SFTON P0306
MOVL C00045 BC00045 V=500.0 PL=0
SFTOF
MOVL C00046 BC00046 V=500.0
MOVL C00047 BC00047 V=500.0
MOVL C00048 BC00048 V=500.0
MOVJ C00049 BC00049 VJ=30.00
MOVL C00050 BC00050 V=500.0
MOVL C00051 BC00051 V=500.0
'------------------------
'W65.20
'------------------------
MOVL C00052 BC00052 V=500.0
MOVL C00053 BC00053 V=333.3 PL=0
REFP 3 C00054 BC00054
CALL JOB:SEARCH-R1
SET P0307 P0006
SFTON P0307
MOVL C00055 BC00055 V=333.3 PL=0
REFP 3 C00056 BC00056
CALL JOB:SEARCH-R1
SET P0307 P0006
SFTON P0307
MOVL C00057 BC00057 V=500.0 PL=0
SFTOF
'------------------------
'W65.23
'------------------------
MOVL C00058 BC00058 V=500.0
MOVL C00059 BC00059 V=333.3 PL=0
REFP 3 C00060 BC00060
CALL JOB:SEARCH-R1
SET P0308 P0006
SFTON P0308
MOVL C00061 BC00061 V=333.3 PL=0
REFP 3 C00062 BC00062
CALL JOB:SEARCH-R1
SET P0308 P0006
SFTON P0308
MOVL C00063 BC00063 V=500.0 PL=0
SFTOF
'------------------------
'W65.25
'------------------------
MOVL C00064 BC00064 V=500.0
MOVL C00065 BC00065 V=333.3 PL=0
REFP 3 C00066 BC00066
CALL JOB:SEARCH-R1
SET P0309 P0006
SFTON P0309
MOVL C00067 BC00067 V=333.3 PL=0
REFP 3 C00068 BC00068
CALL JOB:SEARCH-R1
SET P0309 P0006
SFTON P0309
MOVL C00069 BC00069 V=500.0 PL=0
SFTOF
MOVL C00070 BC00070 V=500.0
MOVL C00071 BC00071 V=500.0
MOVL C00072 BC00072 V=500.0
MOVL C00073 BC00073 V=500.0
MOVL C00074 BC00074 V=500.0
MOVL C00075 BC00075 V=250.0
MOVL C00076 BC00076 V=500.0
MOVL C00077 BC00077 V=500.0
MOVL C00078 BC00078 V=83.3
'------------------------
'W65.28
'------------------------
MOVL C00079 BC00079 V=500.0
MOVL C00080 BC00080 V=333.3 PL=0
REFP 3 C00081 BC00081
CALL JOB:SEARCH-R1
SET P0310 P0006
SFTON P0310
MOVL C00082 BC00082 V=333.3 PL=0
REFP 3 C00083 BC00083
CALL JOB:SEARCH-R1
SET P0310 P0006
SFTON P0310
MOVL C00084 BC00084 V=333.3 PL=0
SFTOF
'------------------------
'W65.30
'------------------------
MOVL C00085 BC00085 V=500.0
MOVL C00086 BC00086 V=333.3 PL=0
REFP 3 C00087 BC00087
CALL JOB:SEARCH-R1
SET P0311 P0006
SFTON P0311
MOVL C00088 BC00088 V=333.3 PL=0
REFP 3 C00089 BC00089
CALL JOB:SEARCH-R1
SET P0311 P0006
SFTON P0311
MOVL C00090 BC00090 V=333.3 PL=0
SFTOF
MOVL C00091 BC00091 V=500.0
MOVL C00092 BC00092 V=500.0
MOVJ C00093 BC00093 VJ=30.00
MOVJ C00094 BC00094 VJ=30.00
MOVJ C00095 BC00095 VJ=30.00
MOVJ C00096 BC00096 VJ=30.00
'------------------------
'W251A
'------------------------
MOVL C00097 BC00097 V=333.3 PL=0
REFP 3 C00098 BC00098
CALL JOB:SEARCH-R1
IMOV P0058 V=16.7
SET P0350 P0006
SFTON P0350
REFP 3 C00099 BC00099
CALL JOB:SEARCH-R1
SET P0350 P0006
SFTON P0350
MOVL C00100 BC00100 V=500.0 PL=0
SFTOF
MOVL C00101 BC00101 V=500.0
MOVL C00102 BC00102 V=500.0
MOVL C00103 BC00103 V=333.3 PL=0
REFP 3 C00104 BC00104
CALL JOB:SEARCH-R1
IMOV P0058 V=16.7
SET P0349 P0006
SFTON P0349
REFP 3 C00105 BC00105
CALL JOB:SEARCH-R1
SET P0349 P0006
SFTON P0349
MOVL C00106 BC00106 V=500.0 PL=0
SFTOF
'------------------------
'W254A P
'------------------------
MOVJ C00107 BC00107 VJ=30.00
MOVL C00108 BC00108 V=333.3 PL=0
REFP 3 C00109 BC00109
CALL JOB:SEARCH-R1
IMOV P0058 V=16.7
SET P0351 P0006
SFTON P0351
REFP 3 C00110 BC00110
CALL JOB:SEARCH-R1
SET P0351 P0006
SFTON P0351
MOVL C00111 BC00111 V=500.0 PL=0
SFTOF
'------------------------
'W254A L
'------------------------
MOVJ C00112 BC00112 VJ=30.00
MOVL C00113 BC00113 V=333.3 PL=0
REFP 3 C00114 BC00114
CALL JOB:SEARCH-R1
IMOV P0058 V=16.7
SET P0352 P0006
SFTON P0352
REFP 3 C00115 BC00115
CALL JOB:SEARCH-R1
SET P0352 P0006
SFTON P0352
MOVL C00116 BC00116 V=500.0 PL=0
SFTOF
'------------------------
'W250A P
'------------------------
MOVJ C00117 BC00117 VJ=30.00
MOVL C00118 BC00118 V=333.3 PL=0
REFP 3 C00119 BC00119
CALL JOB:SEARCH-R1
IMOV P0058 V=16.7
SET P0353 P0006
SFTON P0353
REFP 3 C00120 BC00120
CALL JOB:SEARCH-R1
SET P0353 P0006
SFTON P0353
MOVL C00121 BC00121 V=500.0 PL=0
SFTOF
'------------------------
'W250A L
'------------------------
MOVJ C00122 BC00122 VJ=30.00
MOVL C00123 BC00123 V=333.3 PL=0
REFP 3 C00124 BC00124
CALL JOB:SEARCH-R1
IMOV P0058 V=16.7
SET P0354 P0006
SFTON P0354
REFP 3 C00125 BC00125
CALL JOB:SEARCH-R1
SET P0354 P0006
SFTON P0354
MOVL C00126 BC00126 V=500.0 PL=0
SFTOF
'------------------------
'W253A P
'------------------------
MOVJ C00127 BC00127 VJ=30.00
MOVL C00128 BC00128 V=333.3 PL=0
REFP 3 C00129 BC00129
CALL JOB:SEARCH-R1
IMOV P0058 V=16.7
SET P0355 P0006
SFTON P0355
REFP 3 C00130 BC00130
CALL JOB:SEARCH-R1
SET P0355 P0006
SFTON P0355
MOVL C00131 BC00131 V=333.3 PL=0
SFTOF
'------------------------
'W253A L
'------------------------
MOVJ C00132 BC00132 VJ=30.00
MOVL C00133 BC00133 V=333.3 PL=0
REFP 3 C00134 BC00134
CALL JOB:SEARCH-R1
IMOV P0058 V=16.7
SET P0356 P0006
SFTON P0356
REFP 3 C00135 BC00135
CALL JOB:SEARCH-R1
SET P0356 P0006
SFTON P0356
MOVL C00136 BC00136 V=500.0 PL=0
SFTOF
'------------------------
'W256A P
'------------------------
MOVJ C00137 BC00137 VJ=30.00
MOVL C00138 BC00138 V=333.3 PL=0
REFP 3 C00139 BC00139
CALL JOB:SEARCH-R1
IMOV P0058 V=16.7
SET P0357 P0006
SFTON P0357
REFP 3 C00140 BC00140
CALL JOB:SEARCH-R1
SET P0357 P0006
SFTON P0357
MOVL C00141 BC00141 V=500.0 PL=0
SFTOF
'------------------------
'W256A L
'------------------------
MOVJ C00142 BC00142 VJ=30.00
MOVL C00143 BC00143 V=333.3 PL=0
REFP 3 C00144 BC00144
CALL JOB:SEARCH-R1
IMOV P0058 V=16.7
SET P0358 P0006
SFTON P0358
REFP 3 C00145 BC00145
CALL JOB:SEARCH-R1
SET P0358 P0006
SFTON P0358
MOVL C00146 BC00146 V=500.0 PL=0
SFTOF
'------------------------
'W252A P
'------------------------
MOVL C00147 BC00147 V=500.0
MOVL C00148 BC00148 V=333.3 PL=0
REFP 3 C00149 BC00149
CALL JOB:SEARCH-R1
IMOV P0058 V=16.7
SET P0359 P0006
SFTON P0359
REFP 3 C00150 BC00150
CALL JOB:SEARCH-R1
SET P0359 P0006
SFTON P0359
MOVL C00151 BC00151 V=333.3 PL=0
SFTOF
'------------------------
'W252A L
'------------------------
MOVL C00152 BC00152 V=500.0
MOVL C00153 BC00153 V=333.3 PL=0
REFP 3 C00154 BC00154
CALL JOB:SEARCH-R1
IMOV P0058 V=16.7
SET P0360 P0006
SFTON P0360
REFP 3 C00155 BC00155
CALL JOB:SEARCH-R1
SET P0360 P0006
SFTON P0360
MOVL C00156 BC00156 V=500.0 PL=0
SFTOF
'------------------------
'W255A
'------------------------
MOVL C00157 BC00157 V=500.0
MOVL C00158 BC00158 V=333.3 PL=0
REFP 3 C00159 BC00159
CALL JOB:SEARCH-R1
IMOV P0058 V=16.7
SET P0361 P0006
SFTON P0361
REFP 3 C00160 BC00160
CALL JOB:SEARCH-R1
SET P0361 P0006
SFTON P0361
MOVL C00161 BC00161 V=500.0 PL=0
SFTOF
MOVL C00162 BC00162 V=500.0
MOVJ C00163 BC00163 VJ=50.00
MOVJ C00164 BC00164 VJ=50.00
MOVJ C00165 BC00165 VJ=50.00
COMM MOVJ C00166 BC00166 VJ=30.00
COMM MOVJ C00167 BC00167 VJ=30.00
COMM MOVJ C00168 BC00168 VJ=30.00
COMM MOVJ C00169 BC00169 VJ=50.00
COMM 'COMMENT
COMM MOVJ C00170 BC00170 VJ=50.00
COMM MOVJ C00171 BC00171 VJ=30.00
COMM GETE D040 P0400 (1)
COMM GETE D041 P0400 (2)
COMM GETE D042 P0400 (3)
COMM SETE P0401 (1) D040
COMM SETE P0401 (2) D041
COMM SETE P0401 (3) D042
COMM GETE D040 P0400 (1)
COMM GETE D041 P0400 (2)
COMM GETE D042 P0400 (3)
COMM SETE P0402 (1) D040
COMM SETE P0402 (2) D041
COMM SETE P0402 (3) D042
COMM MOVL C00172 BC00172 V=333.3
COMM MOVL C00173 BC00173 V=333.3
COMM MOVL C00174 BC00174 V=333.3
COMM MOVL C00175 BC00175 V=333.3
COMM '------------------------
COMM 'W61.5
COMM '------------------------
COMM MOVL C00176 BC00176 V=66.7 PL=0
COMM REFP 3 C00177 BC00177
COMM CALL JOB:SEARCH-R1
COMM SET P0401 P0006
COMM SFTON P0401
COMM MOVL C00178 BC00178 V=66.7 PL=0
COMM REFP 3 C00179 BC00179
COMM CALL JOB:SEARCH-R1
COMM SET P0401 P0006
COMM SFTON P0401
COMM MOVL C00180 BC00180 V=66.7 PL=0
COMM SFTOF
COMM MOVL C00181 BC00181 V=333.3
COMM MOVL C00182 BC00182 V=333.3
COMM '------------------------
COMM 'W61.7
COMM '------------------------
COMM MOVL C00183 BC00183 V=333.3
COMM MOVL C00184 BC00184 V=66.7 PL=0
COMM REFP 3 C00185 BC00185
COMM CALL JOB:SEARCH-R1
COMM SET P0402 P0006
COMM SFTON P0402
COMM MOVL C00186 BC00186 V=66.7 PL=0
COMM REFP 3 C00187 BC00187
COMM CALL JOB:SEARCH-R1
COMM SET P0402 P0006
COMM SFTON P0402
COMM MOVL C00188 BC00188 V=66.7 PL=0
COMM SFTOF
COMM '------------------------
COMM 'W61.10
COMM '------------------------
COMM MOVL C00189 BC00189 V=500.0
COMM MOVL C00190 BC00190 V=166.7 PL=0
COMM REFP 3 C00191 BC00191
COMM CALL JOB:SEARCH-R1
COMM SET P0403 P0006
COMM SFTON P0403
COMM MOVL C00192 BC00192 V=166.7 PL=0
COMM REFP 3 C00193 BC00193
COMM CALL JOB:SEARCH-R1
COMM SET P0403 P0006
COMM SFTON P0403
COMM MOVL C00194 BC00194 V=500.0 PL=0
COMM SFTOF
COMM '------------------------
COMM 'W61.12
COMM '------------------------
COMM MOVL C00195 BC00195 V=500.0
COMM MOVL C00196 BC00196 V=166.7 PL=0
COMM REFP 3 C00197 BC00197
COMM CALL JOB:SEARCH-R1
COMM SET P0404 P0006
COMM SFTON P0404
COMM MOVL C00198 BC00198 V=166.7 PL=0
COMM REFP 3 C00199 BC00199
COMM CALL JOB:SEARCH-R1
COMM SET P0404 P0006
COMM SFTON P0404
COMM MOVL C00200 BC00200 V=500.0 PL=0
COMM SFTOF
COMM '------------------------
COMM 'W61.15
COMM '------------------------
COMM MOVL C00201 BC00201 V=500.0
COMM MOVL C00202 BC00202 V=166.7 PL=0
COMM REFP 3 C00203 BC00203
COMM CALL JOB:SEARCH-R1
COMM SET P0405 P0006
COMM SFTON P0405
COMM MOVL C00204 BC00204 V=166.7 PL=0
COMM REFP 3 C00205 BC00205
COMM CALL JOB:SEARCH-R1
COMM SET P0405 P0006
COMM SFTON P0405
COMM MOVL C00206 BC00206 V=500.0 PL=0
COMM SFTOF
COMM MOVL C00207 BC00207 V=500.0
COMM SFTOF
COMM GETE D040 P0405 (1)
COMM GETE D041 P0405 (2)
COMM GETE D042 P0405 (3)
COMM SETE P0406 (1) D040
COMM SETE P0406 (2) D041
COMM SETE P0406 (3) D042
COMM '------------------------
COMM 'W61.17
COMM '------------------------
COMM MOVL C00208 BC00208 V=333.3
COMM MOVL C00209 BC00209 V=66.7 PL=0
COMM REFP 3 C00210 BC00210
COMM CALL JOB:SEARCH-R1
COMM SET P0406 P0006
COMM SFTON P0406
COMM MOVL C00211 BC00211 V=66.7 PL=0
COMM REFP 3 C00212 BC00212
COMM CALL JOB:SEARCH-R1
COMM SET P0406 P0006
COMM SFTON P0406
COMM MOVL C00213 BC00213 V=66.7 PL=0
COMM SFTOF
COMM MOVL C00214 BC00214 V=333.3
COMM MOVL C00215 BC00215 V=333.3
COMM MOVJ C00216 BC00216 VJ=30.00
COMM MOVJ C00217 BC00217 VJ=50.00
COMM MOVL C00218 BC00218 V=666.7
COMM '------------------------
COMM 'W61.20
COMM '------------------------
COMM MOVL C00219 BC00219 V=500.0
COMM MOVL C00220 BC00220 V=166.7 PL=0
COMM REFP 3 C00221 BC00221
COMM CALL JOB:SEARCH-R1
COMM SET P0407 P0006
COMM SFTON P0407
COMM MOVL C00222 BC00222 V=166.7 PL=0
COMM REFP 3 C00223 BC00223
COMM CALL JOB:SEARCH-R1
COMM SET P0407 P0006
COMM SFTON P0407
COMM MOVL C00224 BC00224 V=500.0 PL=0
COMM SFTOF
COMM '------------------------
COMM 'W61.23
COMM '------------------------
COMM MOVL C00225 BC00225 V=500.0
COMM MOVL C00226 BC00226 V=166.7 PL=0
COMM REFP 3 C00227 BC00227
COMM CALL JOB:SEARCH-R1
COMM SET P0408 P0006
COMM SFTON P0408
COMM MOVL C00228 BC00228 V=166.7 PL=0
COMM REFP 3 C00229 BC00229
COMM CALL JOB:SEARCH-R1
COMM SET P0408 P0006
COMM SFTON P0408
COMM MOVL C00230 BC00230 V=500.0 PL=0
COMM SFTOF
COMM '------------------------
COMM 'W61.25
COMM '------------------------
COMM MOVL C00231 BC00231 V=500.0
COMM MOVL C00232 BC00232 V=166.7 PL=0
COMM REFP 3 C00233 BC00233
COMM CALL JOB:SEARCH-R1
COMM SET P0409 P0006
COMM SFTON P0409
COMM MOVL C00234 BC00234 V=166.7 PL=0
COMM REFP 3 C00235 BC00235
COMM CALL JOB:SEARCH-R1
COMM SET P0409 P0006
COMM SFTON P0409
COMM MOVL C00236 BC00236 V=500.0 PL=0
COMM SFTOF
COMM MOVL C00237 BC00237 V=500.0
COMM MOVL C00238 BC00238 V=500.0
COMM MOVJ C00239 BC00239 VJ=50.00
COMM MOVL C00240 BC00240 V=666.7
COMM GETE D040 P0409 (1)
COMM GETE D041 P0409 (2)
COMM GETE D042 P0409 (3)
COMM SETE P0410 (1) D040
COMM SETE P0410 (2) D041
COMM SETE P0410 (3) D042
COMM '------------------------
COMM 'W61.30
COMM '------------------------
COMM MOVL C00241 BC00241 V=500.0
COMM MOVL C00242 BC00242 V=166.7 PL=0
COMM REFP 3 C00243 BC00243
COMM CALL JOB:SEARCH-R1
COMM SET P0411 P0006
COMM SFTON P0411
COMM MOVL C00244 BC00244 V=166.7 PL=0
COMM REFP 3 C00245 BC00245
COMM CALL JOB:SEARCH-R1
COMM SET P0411 P0006
COMM SFTON P0411
COMM MOVL C00246 BC00246 V=500.0 PL=0
COMM SFTOF
COMM MOVL C00247 BC00247 V=666.7
COMM MOVJ C00248 BC00248 VJ=30.00
MOVJ C00249 BC00249 VJ=50.00
IFTHENEXP OT#(1457)=ON ANDEXP OT#(1441)=OFF
	 CALL JOB:TWIN_FRONT_SEARCH_90ST-2_5340
ENDIF
IFTHENEXP OT#(1457)=OFF ANDEXP OT#(1441)=ON
	 CALL JOB:FRONT_SEARCH_90ST-2_5340
ENDIF
MOVJ C00250 BC00250 VJ=50.00
MOVJ C00251 BC00251 VJ=40.00
MOVJ C00252 BC00252 VJ=30.00
MOVL C00253 BC00253 V=666.7
MOVJ C00254 BC00254 VJ=40.00
'------------------------
'W65.3
'------------------------
SFTON P0300
MOVL C00255 BC00255 V=500.0
MOVL C00256 BC00256 V=333.3 PL=0
MACRO1 MJ#(0) ARGF10
ARCON
MOVL C00257 BC00257 V=10.8
ARCOF
MOVL C00258 BC00258 V=166.7
SFTOF
'------------------------
'W65.5
'------------------------
SFTON P0301
MOVL C00259 BC00259 V=333.3
MOVL C00260 BC00260 V=133.3 PL=0
MACRO1 MJ#(0) ARGF10
ARCON
MOVL C00261 BC00261 V=10.8
ARCOF
MOVL C00262 BC00262 V=166.7
SFTOF
MOVL C00263 BC00263 V=500.0
MOVL C00264 BC00264 V=333.3
MOVJ C00265 BC00265 VJ=25.00
MOVJ C00266 BC00266 VJ=50.00
'::::::::::::::::::::::::::::::::
'::::::::::::::::::::::::::::::::
'::::::::::::::::::::::::::::::::
'::::::::::::::::::::::::::::::::
'::::::::::::::::::::::::::::::::
COMM MOVJ C00267 BC00267 VJ=50.00
COMM MOVJ C00268 BC00268 VJ=50.00
COMM MOVJ C00269 BC00269 VJ=50.00
COMM MOVJ C00270 BC00270 VJ=50.00
COMM MOVJ C00271 BC00271 VJ=20.00
COMM '------------------------
COMM 'W61.3
COMM '------------------------
COMM SFTON P0400
COMM MOVL C00272 BC00272 V=333.3
COMM MOVL C00273 BC00273 V=66.7 PL=0
COMM MACRO1 MJ#(0) ARGF9
COMM ARCOF
COMM SFTOF
COMM 'BELKA PRZEJAZD
COMM MOVJ C00274 BC00274 VJ=25.00
COMM MOVJ C00275 BC00275 VJ=50.00
COMM MOVL C00276 BC00276 V=500.0
COMM MOVL C00277 BC00277 V=500.0
COMM '------------------------
COMM 'W61.5
COMM '------------------------
COMM SFTON P0401
COMM MOVL C00278 BC00278 V=333.3
COMM MOVL C00279 BC00279 V=133.3 PL=0
COMM MACRO1 MJ#(0) ARGF24
COMM ARCON
COMM MOVL C00280 BC00280 V=7.5
COMM ARCOF
COMM MOVL C00281 BC00281 V=250.0
COMM SFTOF
COMM MOVL C00282 BC00282 V=333.3
COMM MOVJ C00283 BC00283 VJ=35.00
COMM MOVJ C00284 BC00284 VJ=50.00
COMM MOVJ C00285 BC00285 VJ=50.00
COMM MOVJ C00286 BC00286 VJ=50.00
MOVJ C00287 BC00287 VJ=50.00
MOVJ C00288 BC00288 VJ=50.00
MOVJ C00289 BC00289 VJ=50.00
'------------------------
'W250A
'------------------------
SFTON P0354
MOVL C00290 BC00290 V=333.3
MOVL C00291 BC00291 V=133.3 PL=0
MACRO1 MJ#(0) ARGF9
ARCON
SFTOF
SFTON P0353
MOVL C00292 BC00292 V=11.7
ARCOF
MOVL C00293 BC00293 V=166.7
SFTOF
MOVJ C00294 BC00294 VJ=50.00
MOVJ C00295 BC00295 VJ=50.00
MOVJ C00296 BC00296 VJ=50.00
MOVJ C00297 BC00297 VJ=50.00
MOVJ C00298 BC00298 VJ=50.00
MOVJ C00299 BC00299 VJ=20.00
MOVJ C00300 BC00300 VJ=10.00
'------------------------
'W65.7
'------------------------
SFTON P0302
'MOTOSIM PULSE LIMIT
MOVL C00301 BC00301 V=500.0
MOVL C00302 BC00302 V=133.3 PL=0
MACRO1 MJ#(0) ARGF10
ARCON
MOVL C00303 BC00303 V=10.8
ARCOF
MOVL C00304 BC00304 V=250.0
SFTOF
'------------------------
'W65.10
'------------------------
SFTON P0303
MOVL C00305 BC00305 V=500.0
MOVL C00306 BC00306 V=166.7 PL=0
ARCON
MOVL C00307 BC00307 V=10.8
ARCOF
MOVL C00308 BC00308 V=166.7
SFTOF
SFTOF
MOVL C00309 BC00309 V=333.3
MOVL C00310 BC00310 V=500.0
MOVJ C00311 BC00311 VJ=50.00
MOVJ C00312 BC00312 VJ=30.00
MOVJ C00313 BC00313 VJ=50.00
MOVJ C00314 BC00314 VJ=50.00
COMM '::::::::::::::::::::::::::::::::
COMM '::::::::::::::::::::::::::::::::
COMM '------------------------
COMM 'W61.7
COMM '------------------------
COMM '::::::::::::::::::::::::::::::::
COMM '::::::::::::::::::::::::::::::::
COMM MOVJ C00315 BC00315 VJ=50.00
COMM MOVJ C00316 BC00316 VJ=35.00
COMM SFTON P0402
COMM MOVL C00317 BC00317 V=333.3
COMM MOVL C00318 BC00318 V=133.3 PL=0
COMM MACRO1 MJ#(0) ARGF24
COMM ARCON
COMM MOVL C00319 BC00319 V=7.5
COMM ARCOF
COMM MOVL C00320 BC00320 V=166.7
COMM SFTOF
COMM MOVL C00321 BC00321 V=500.0
COMM MOVL C00322 BC00322 V=500.0
COMM MOVJ C00323 BC00323 VJ=50.00
COMM '------------------------
COMM 'W61.10
COMM '------------------------
COMM SFTON P0403
COMM MOVL C00324 BC00324 V=333.3
COMM MOVL C00325 BC00325 V=133.3 PL=0
COMM MACRO1 MJ#(0) ARGF24
COMM ARCON
COMM MOVL C00326 BC00326 V=7.5
COMM ARCOF
COMM MOVL C00327 BC00327 V=166.7
COMM SFTOF
COMM MOVL C00328 BC00328 V=333.3
COMM MOVJ C00329 BC00329 VJ=35.00
COMM MOVJ C00330 BC00330 VJ=50.00
COMM MOVJ C00331 BC00331 VJ=50.00
COMM '::::::::::::::::::::::::
COMM '::::::::::::::::::::::::
COMM '::::::::::::::::::::::::
COMM '::::::::::::::::::::::::
COMM '::::::::::::::::::::::::
COMM '::::::::::::::::::::::::
COMM '::::::::::::::::::::::::
MOVJ C00332 BC00332 VJ=50.00
MOVJ C00333 BC00333 VJ=50.00
MOVJ C00334 BC00334 VJ=50.00
'------------------------
'W214A
'------------------------
SFTON P0350
MOVL C00335 BC00335 V=333.3
MOVL C00336 BC00336 V=333.3
MOVL C00337 BC00337 V=133.3 PL=0
MACRO1 MJ#(0) ARGF9
ARCON
SFTOF
SFTON P0349
MOVL C00338 BC00338 V=11.7
MOVL C00339 BC00339 V=11.7
ARCOF
MOVL C00340 BC00340 V=250.0
SFTOF
MOVJ C00341 BC00341 VJ=50.00
MOVJ C00342 BC00342 VJ=50.00
MOVJ C00343 BC00343 VJ=50.00
MOVJ C00344 BC00344 VJ=50.00
MOVJ C00345 BC00345 VJ=50.00
MOVJ C00346 BC00346 VJ=50.00
MOVJ C00347 BC00347 VJ=20.00
'------------------------
'W65.12
'------------------------
SFTON P0304
MOVL C00348 BC00348 V=333.3
MOVL C00349 BC00349 V=133.3 PL=0
MACRO1 MJ#(0) ARGF10
ARCON
MOVL C00350 BC00350 V=10.8
ARCOF
MOVL C00351 BC00351 V=166.7
SFTOF
'------------------------
'W65.15
'------------------------
SFTON P0305
MOVL C00352 BC00352 V=333.3
MOVL C00353 BC00353 V=166.7 PL=0
MACRO1 MJ#(0) ARGF10
ARCON
MOVL C00354 BC00354 V=10.8
ARCOF
MOVL C00355 BC00355 V=166.7
SFTOF
MOVL C00356 BC00356 V=333.3
MOVL C00357 BC00357 V=500.0
MOVL C00358 BC00358 V=500.0
MOVJ C00359 BC00359 VJ=50.00
COMM '::::::::::::::::::::::::
COMM '::::::::::::::::::::::::
COMM '::::::::::::::::::::::::
COMM '::::::::::::::::::::::::
COMM '::::::::::::::::::::::::
COMM '::::::::::::::::::::::::
COMM '::::::::::::::::::::::::
COMM MOVJ C00360 BC00360 VJ=50.00
COMM MOVJ C00361 BC00361 VJ=50.00
COMM '::::::::::::::::::::::::::::::::
COMM '::::::::::::::::::::::::::::::::
COMM '------------------------
COMM 'W61.12
COMM '------------------------
COMM '::::::::::::::::::::::::::::::::
COMM '::::::::::::::::::::::::::::::::
COMM SFTON P0404
COMM MOVJ C00362 BC00362 VJ=50.00
COMM MOVL C00363 BC00363 V=333.3
COMM MOVL C00364 BC00364 V=333.3
COMM MOVL C00365 BC00365 V=166.7 PL=0
COMM MACRO1 MJ#(0) ARGF24
COMM ARCON
COMM MOVL C00366 BC00366 V=7.5
COMM ARCOF
COMM MOVL C00367 BC00367 V=166.7
COMM SFTOF
COMM MOVL C00368 BC00368 V=333.3
COMM MOVL C00369 BC00369 V=333.3
COMM '------------------------
COMM 'W61.15
COMM '------------------------
COMM SFTON P0405
COMM MOVL C00370 BC00370 V=333.3
COMM MOVL C00371 BC00371 V=166.7 PL=0
COMM MACRO1 MJ#(0) ARGF24
COMM ARCON
COMM MOVL C00372 BC00372 V=7.5
COMM ARCOF
COMM MOVL C00373 BC00373 V=166.7
COMM SFTOF
COMM MOVJ C00374 BC00374 VJ=50.00
COMM MOVJ C00375 BC00375 VJ=50.00
COMM MOVJ C00376 BC00376 VJ=50.00
COMM '::::::::::::::::::::::::
COMM '::::::::::::::::::::::::
COMM '::::::::::::::::::::::::
COMM '::::::::::::::::::::::::
COMM '::::::::::::::::::::::::
COMM '::::::::::::::::::::::::
COMM '::::::::::::::::::::::::
MOVJ C00377 BC00377 VJ=50.00
MOVJ C00378 BC00378 VJ=50.00
'------------------------
'W252A
'------------------------
SFTON P0359
MOVL C00379 BC00379 V=500.0
MOVL C00380 BC00380 V=166.7 PL=0
MACRO1 MJ#(0) ARGF9
ARCON
SFTOF
SFTON P0358
MOVL C00381 BC00381 V=11.7
ARCOF
MOVL C00382 BC00382 V=250.0
SFTOF
MOVJ C00383 BC00383 VJ=50.00
MOVJ C00384 BC00384 VJ=80.00
COMM MOVJ C00385 BC00385 VJ=80.00
COMM MOVJ C00386 BC00386 VJ=50.00
COMM MOVJ C00387 BC00387 VJ=50.00
COMM MOVJ C00388 BC00388 VJ=25.00
'::::::::::::::::::::::::
'::::::::::::::::::::::::
'::::::::::::::::::::::::
'::::::::::::::::::::::::
'::::::::::::::::::::::::
'::::::::::::::::::::::::
'::::::::::::::::::::::::
'::::::::::::::::::::::::::::::::
'::::::::::::::::::::::::::::::::
'------------------------
'W61.17
'------------------------
'::::::::::::::::::::::::::::::::
'::::::::::::::::::::::::::::::::
COMM SFTON P0406
COMM MOVJ C00389 BC00389 VJ=10.00
COMM MOVL C00390 BC00390 V=150.0
COMM MOVL C00391 BC00391 V=66.7 PL=0
COMM MACRO1 MJ#(0) ARGF24
COMM ARCON
COMM MOVL C00392 BC00392 V=6.7
COMM ARCOF
COMM MOVL C00393 BC00393 V=83.3
COMM SFTOF
COMM '------------------------
COMM 'W253A
COMM '------------------------
COMM MOVJ C00394 BC00394 VJ=50.00
MOVJ C00395 BC00395 VJ=50.00
SFTON P0356
MOVL C00396 BC00396 V=333.3
MOVL C00397 BC00397 V=333.3
MOVL C00398 BC00398 V=166.7 PL=0
MACRO1 MJ#(0) ARGF9
ARCON
SFTOF
SFTON P0355
MOVL C00399 BC00399 V=11.7
ARCOF
MOVL C00400 BC00400 V=250.0
SFTOF
MOVJ C00401 BC00401 VJ=50.00
MOVJ C00402 BC00402 VJ=50.00
MOVJ C00403 BC00403 VJ=80.00
MOVJ C00404 BC00404 VJ=80.00
MOVJ C00405 BC00405 VJ=50.00
MOVJ C00406 BC00406 VJ=50.00
MOVJ C00407 BC00407 VJ=50.00
MOVJ C00408 BC00408 VJ=30.00
MOVJ C00409 BC00409 VJ=30.00
'------------------------
'W65.20
'------------------------
SFTON P0307
MOVL C00410 BC00410 V=333.3
MOVL C00411 BC00411 V=166.7
MOVL C00412 BC00412 V=166.7 PL=0
MACRO1 MJ#(0) ARGF10
ARCON
MOVL C00413 BC00413 V=10.8
ARCOF
MOVL C00414 BC00414 V=500.0
MOVL C00415 BC00415 V=500.0
MOVL C00416 BC00416 V=166.7
ARCON
MOVL C00417 BC00417 V=10.8
ARCOF
MOVL C00418 BC00418 V=250.0
SFTOF
MOVL C00419 BC00419 V=333.3
MOVL C00420 BC00420 V=333.3
MOVL C00421 BC00421 V=333.3
MOVJ C00422 BC00422 VJ=50.00
MOVJ C00423 BC00423 VJ=50.00
MOVJ C00424 BC00424 VJ=50.00
MOVJ C00425 BC00425 VJ=50.00
COMM '::::::::::::::::::::::::
COMM '::::::::::::::::::::::::
COMM '::::::::::::::::::::::::
COMM '::::::::::::::::::::::::
COMM '::::::::::::::::::::::::
COMM '::::::::::::::::::::::::
COMM '::::::::::::::::::::::::
COMM MOVJ C00426 BC00426 VJ=80.00
COMM MOVJ C00427 BC00427 VJ=50.00
COMM MOVJ C00428 BC00428 VJ=50.00
COMM '::::::::::::::::::::::::::::::::
COMM '::::::::::::::::::::::::::::::::
COMM '------------------------
COMM 'W61.20
COMM '------------------------
COMM '::::::::::::::::::::::::::::::::
COMM '::::::::::::::::::::::::::::::::
COMM SFTON P0407
COMM MOVL C00429 BC00429 V=333.3
COMM MOVL C00430 BC00430 V=166.7
COMM MOVL C00431 BC00431 V=133.3 PL=0
COMM MACRO1 MJ#(0) ARGF24
COMM ARCON
COMM MOVL C00432 BC00432 V=7.5
COMM ARCOF
COMM MOVL C00433 BC00433 V=166.7
COMM SFTOF
COMM SFTON P0407
COMM MOVL C00434 BC00434 V=166.7
COMM MOVL C00435 BC00435 V=133.3 PL=0
COMM MACRO1 MJ#(0) ARGF24
COMM ARCON
COMM MOVL C00436 BC00436 V=7.5
COMM ARCOF
COMM MOVL C00437 BC00437 V=166.7
COMM SFTOF
COMM '::::::::::::::::::::::::
COMM '::::::::::::::::::::::::
COMM '::::::::::::::::::::::::
COMM '::::::::::::::::::::::::
COMM '::::::::::::::::::::::::
COMM MOVJ C00438 BC00438 VJ=50.00
COMM MOVJ C00439 BC00439 VJ=50.00
COMM MOVJ C00440 BC00440 VJ=50.00
COMM MOVJ C00441 BC00441 VJ=50.00
COMM '------------------------
COMM 'W254A
COMM '------------------------
MOVJ C00442 BC00442 VJ=50.00
MOVJ C00443 BC00443 VJ=50.00
SFTON P0352
MOVL C00444 BC00444 V=500.0
MOVL C00445 BC00445 V=500.0
MOVL C00446 BC00446 V=166.7 PL=0
MACRO1 MJ#(0) ARGF9
ARCON
SFTOF
SFTON P0351
MOVL C00447 BC00447 V=11.7
ARCOF
MOVL C00448 BC00448 V=333.3
SFTOF
COMM MOVJ C00449 BC00449 VJ=80.00
COMM MOVJ C00450 BC00450 VJ=80.00
COMM MOVJ C00451 BC00451 VJ=80.00
COMM MOVJ C00452 BC00452 VJ=80.00
COMM MOVJ C00453 BC00453 VJ=50.00
MOVJ C00454 BC00454 VJ=50.00
MOVJ C00455 BC00455 VJ=50.00
MOVJ C00456 BC00456 VJ=50.00
MOVJ C00457 BC00457 VJ=30.00
MOVL C00458 BC00458 V=500.0
'------------------------
'W65.23
'------------------------
SFTON P0308
MOVL C00459 BC00459 V=333.3
MOVL C00460 BC00460 V=166.7
MOVL C00461 BC00461 V=133.3 PL=0
MACRO1 MJ#(0) ARGF10
ARCON
MOVL C00462 BC00462 V=10.8
ARCOF
MOVL C00463 BC00463 V=166.7
SFTOF
'------------------------
'W65.25
'------------------------
SFTON P0309
MOVL C00464 BC00464 V=500.0
MOVL C00465 BC00465 V=133.3 PL=0
ARCON
MOVL C00466 BC00466 V=10.8
ARCOF
MOVL C00467 BC00467 V=166.7
SFTOF
MOVL C00468 BC00468 V=500.0
MOVL C00469 BC00469 V=333.3
MOVL C00470 BC00470 V=500.0
MOVL C00471 BC00471 V=333.3
MOVJ C00472 BC00472 VJ=50.00
MOVJ C00473 BC00473 VJ=50.00
MOVJ C00474 BC00474 VJ=50.00
MOVJ C00475 BC00475 VJ=80.00
COMM '::::::::::::::::::::::::
COMM '::::::::::::::::::::::::
COMM '::::::::::::::::::::::::
COMM '::::::::::::::::::::::::
COMM '::::::::::::::::::::::::
COMM '::::::::::::::::::::::::
COMM '::::::::::::::::::::::::
COMM MOVJ C00476 BC00476 VJ=80.00
COMM MOVJ C00477 BC00477 VJ=80.00
COMM MOVJ C00478 BC00478 VJ=50.00
COMM MOVJ C00479 BC00479 VJ=50.00
COMM '::::::::::::::::::::::::::::::::
COMM '::::::::::::::::::::::::::::::::
COMM '------------------------
COMM 'W61.23
COMM '------------------------
COMM '::::::::::::::::::::::::::::::::
COMM '::::::::::::::::::::::::::::::::
COMM SFTON P0408
COMM MOVL C00480 BC00480 V=333.3
COMM MOVL C00481 BC00481 V=166.7
COMM MOVL C00482 BC00482 V=133.3 PL=0
COMM MACRO1 MJ#(0) ARGF24
COMM ARCON
COMM MOVL C00483 BC00483 V=7.5
COMM ARCOF
COMM MOVL C00484 BC00484 V=83.3
COMM SFTOF
COMM '------------------------
COMM 'W61.25
COMM '------------------------
COMM SFTON P0409
COMM MOVL C00485 BC00485 V=333.3
COMM MOVL C00486 BC00486 V=150.0
COMM MOVL C00487 BC00487 V=133.3 PL=0
COMM MACRO1 MJ#(0) ARGF24
COMM ARCON
COMM MOVL C00488 BC00488 V=7.5
COMM ARCOF
COMM MOVL C00489 BC00489 V=166.7
COMM SFTOF
COMM '::::::::::::::::::::::::
COMM '::::::::::::::::::::::::
COMM '::::::::::::::::::::::::
COMM '::::::::::::::::::::::::
COMM '::::::::::::::::::::::::
COMM MOVL C00490 BC00490 V=333.3
COMM MOVJ C00491 BC00491 VJ=50.00
COMM MOVJ C00492 BC00492 VJ=50.00
COMM MOVJ C00493 BC00493 VJ=50.00
COMM MOVJ C00494 BC00494 VJ=50.00
MOVJ C00495 BC00495 VJ=80.00
'------------------------
'W255A
MOVL C00496 BC00496 V=500.0
MOVL C00497 BC00497 V=333.3
SFTON P0361
MOVL C00498 BC00498 V=133.3 PL=0
MACRO1 MJ#(0) ARGF9
ARCON
MOVL C00499 BC00499 V=11.7
ARCOF
MOVL C00500 BC00500 V=250.0
SFTOF
MOVL C00501 BC00501 V=333.3
MOVL C00502 BC00502 V=333.3
MOVL C00503 BC00503 V=500.0
MOVJ C00504 BC00504 VJ=50.00
MOVJ C00505 BC00505 VJ=50.00
MOVJ C00506 BC00506 VJ=80.00
MOVJ C00507 BC00507 VJ=50.00
MOVJ C00508 BC00508 VJ=50.00
MOVL C00509 BC00509 V=333.3
'------------------------
'W31.28
'------------------------
SFTON P0310
MOVL C00510 BC00510 V=333.3
MOVL C00511 BC00511 V=333.3
MOVL C00512 BC00512 V=166.7
COMM MOVL C00513 BC00513 V=66.7 PL=0
COMM MACRO1 MJ#(0) ARGF24
COMM ARCON
COMM MOVL C00514 BC00514 V=8.3
COMM ARCOF
MOVL C00515 BC00515 V=83.3
SFTOF
'------------------------
'W31.30
'------------------------
SFTON P0311
MOVL C00516 BC00516 V=333.3
MOVL C00517 BC00517 V=133.3 PL=0
MACRO1 MJ#(0) ARGF10
ARCON
MOVL C00518 BC00518 V=10.8
ARCOF
MOVL C00519 BC00519 V=166.7
MOVL C00520 BC00520 V=333.3
MOVL C00521 BC00521 V=166.7
ARCON
MOVL C00522 BC00522 V=10.8
ARCOF
MOVL C00523 BC00523 V=166.7
ARCON
MOVL C00524 BC00524 V=10.8
ARCOF
MOVL C00525 BC00525 V=166.7
MOVL C00526 BC00526 V=333.3
SFTOF
MOVL C00527 BC00527 V=500.0
MOVL C00528 BC00528 V=333.3
'::::::::::::::::::::::::
'::::::::::::::::::::::::
'::::::::::::::::::::::::
'::::::::::::::::::::::::
'::::::::::::::::::::::::
'::::::::::::::::::::::::
'::::::::::::::::::::::::
MOVJ C00529 BC00529 VJ=50.00 PL=0
COMM MOVJ C00530 BC00530 VJ=50.00
COMM MOVJ C00531 BC00531 VJ=50.00
COMM '::::::::::::::::::::::::::::::::
COMM '::::::::::::::::::::::::::::::::
COMM '------------------------
COMM 'W61.30
COMM '------------------------
COMM '::::::::::::::::::::::::::::::::
COMM '::::::::::::::::::::::::::::::::
COMM SFTON P0411
COMM MOVL C00532 BC00532 V=333.3
COMM MOVL C00533 BC00533 V=133.3 PL=0
COMM MACRO1 MJ#(0) ARGF24
COMM ARCON
COMM MOVL C00534 BC00534 V=7.5
COMM ARCOF
COMM MOVL C00535 BC00535 V=166.7
COMM SFTOF
COMM MOVL C00536 BC00536 V=500.0
COMM MOVJ C00537 BC00537 VJ=50.00
COMM MOVJ C00538 BC00538 VJ=50.00
COMM MOVJ C00539 BC00539 VJ=50.00
COMM MOVJ C00540 BC00540 VJ=80.00
COMM MOVJ C00541 BC00541 VJ=80.00
COMM '------------------------
COMM 'W256A
COMM '------------------------
MOVJ C00542 BC00542 VJ=80.00
MOVJ C00543 BC00543 VJ=80.00
SFTON P0358
MOVL C00544 BC00544 V=333.3
MOVL C00545 BC00545 V=250.0
MOVL C00546 BC00546 V=166.7 PL=0
MACRO1 MJ#(0) ARGF9
ARCON
SFTOF
SFTON P0357
MOVL C00547 BC00547 V=11.7
ARCOF
MOVL C00548 BC00548 V=333.3
SFTOF
MOVJ C00549 BC00549 VJ=50.00
MOVJ C00550 BC00550 VJ=50.00
MOVJ C00551 BC00551 VJ=80.00
IFTHENEXP OT#(1457)=ON ANDEXP OT#(1441)=OFF
	 CALL JOB:TWIN_FRONT_WELD_90ST-2_5340
ENDIF
IFTHENEXP OT#(1457)=OFF ANDEXP OT#(1441)=ON
	 CALL JOB:FRONT_WELD_90ST-2_5340
ENDIF
CALL JOB:MOVE_OUT_OF_TUNNEL
END
